// TIA Portal V16 export
// export: Created 2025-05-24T14:07:36.0860852Z, ExportSetting WithDefaults, DisplayName Totally Integrated Automation Portal, DisplayVersion V16, DisplayName TIA Portal Version Control Interface, DisplayVersion V16, DisplayName TIA Portal Openness, DisplayVersion V16, DisplayName STEP 7 Professional, DisplayVersion V16, DisplayName STEP 7 Safety, DisplayVersion V16, DisplayName WinCC Advanced, DisplayVersion V16
FUNCTION "6 - Storingsmelding" : Void   // FC8, LAD
TITLE = Warnings
VERSION : 0.1
// This program block is for audible & visual warnings.
// stored: AutoNumber true, IsIECCheckEnabled false, UDAEnableTagReadback false
   VAR_TEMP
      "Wals Sensor Controlled" : Bool;
      "Infeed Sensor Controlled" : Bool;
   END_VAR
   VAR CONSTANT
      "Sensor 2 (option)" : Bool := TRUE;
   END_VAR
   VAR_TEMP   // added for the SCL form of the ladder/FBD networks
      _w1 : Bool;
   END_VAR
BEGIN

REGION Network 1: +MC-21K6:5 - Bel Storing
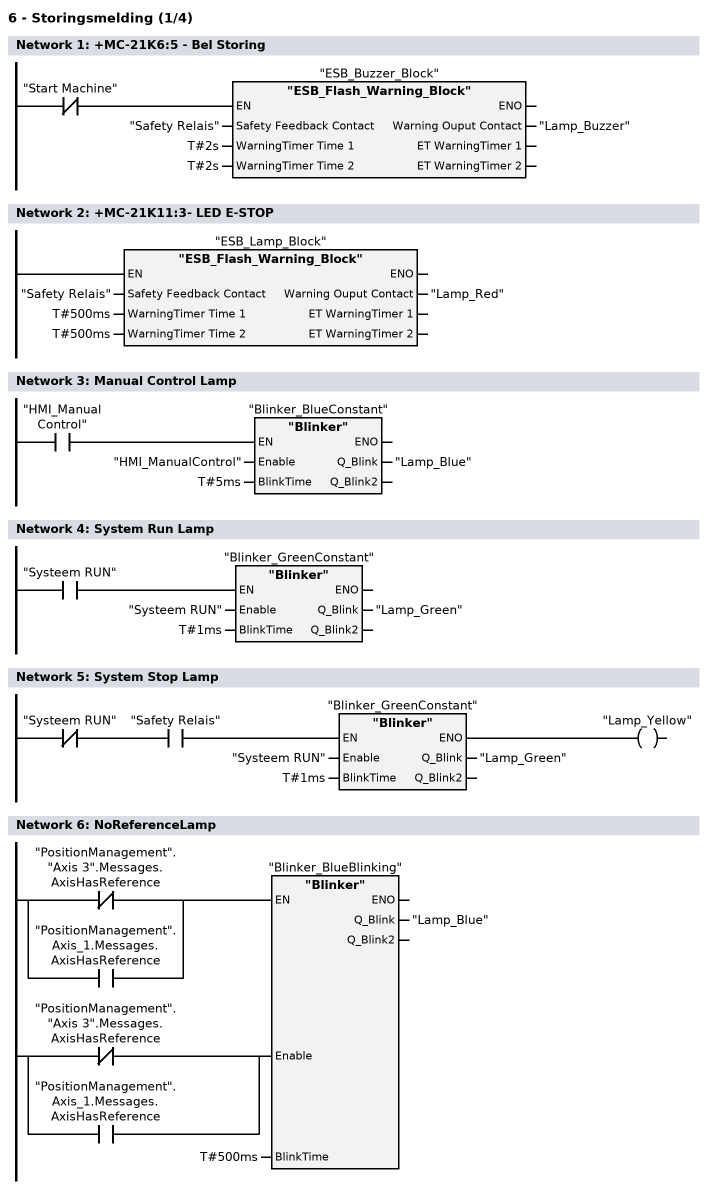
   RUNG wire#powerrail
      I_Contact( "Start Machine" )
      "ESB_Buzzer_Block"("Safety Feedback Contact" := "Safety Relais", "WarningTimer Time 1" := T#2s, "WarningTimer Time 2" := T#2s, "Warning Ouput Contact" => "Lamp_Buzzer", "ET WarningTimer 1" =>, "ET WarningTimer 2" =>)
   END_RUNG
   // the same network as SCL:
   IF NOT "Start Machine" THEN
       "ESB_Buzzer_Block"("Safety Feedback Contact" := "Safety Relais",   // "ESB_Flash_Warning_Block"
                          "WarningTimer Time 1" := T#2s,
                          "WarningTimer Time 2" := T#2s,
                          "Warning Ouput Contact" => "Lamp_Buzzer");
   END_IF;
END_REGION

REGION Network 2: +MC-21K11:3- LED E-STOP
   RUNG wire#powerrail
      "ESB_Lamp_Block"("Safety Feedback Contact" := "Safety Relais", "WarningTimer Time 1" := T#500ms, "WarningTimer Time 2" := T#500ms, "Warning Ouput Contact" => "Lamp_Red", "ET WarningTimer 1" =>, "ET WarningTimer 2" =>)
   END_RUNG
   // the same network as SCL:
   "ESB_Lamp_Block"("Safety Feedback Contact" := "Safety Relais",   // "ESB_Flash_Warning_Block"
                    "WarningTimer Time 1" := T#500ms,
                    "WarningTimer Time 2" := T#500ms,
                    "Warning Ouput Contact" => "Lamp_Red");
END_REGION

REGION Network 3: Manual Control Lamp
   RUNG wire#powerrail
      Contact( "HMI_ManualControl" )
      "Blinker_BlueConstant"(Enable := "HMI_ManualControl", BlinkTime := T#5ms, Q_Blink => "Lamp_Blue", Q_Blink2 =>)
   END_RUNG
   // the same network as SCL:
   IF "HMI_ManualControl" THEN
       "Blinker_BlueConstant"(Enable := "HMI_ManualControl", BlinkTime := T#5ms, Q_Blink => "Lamp_Blue");   // "Blinker"
   END_IF;
END_REGION

REGION Network 4: System Run Lamp
   RUNG wire#powerrail
      Contact( "Systeem RUN" )
      "Blinker_GreenConstant"(Enable := "Systeem RUN", BlinkTime := T#1ms, Q_Blink => "Lamp_Green", Q_Blink2 =>)
   END_RUNG
   // the same network as SCL:
   IF "Systeem RUN" THEN
       "Blinker_GreenConstant"(Enable := "Systeem RUN", BlinkTime := T#1ms, Q_Blink => "Lamp_Green");   // "Blinker"
   END_IF;
END_REGION

REGION Network 5: System Stop Lamp
   RUNG wire#powerrail
      I_Contact( "Systeem RUN" )
      Contact( "Safety Relais" )
      "Blinker_GreenConstant"(Enable := "Systeem RUN", BlinkTime := T#1ms, Q_Blink => "Lamp_Green", Q_Blink2 =>)
      Coil( "Lamp_Yellow" )
   END_RUNG
   // the same network as SCL:
   "Blinker_GreenConstant"(EN := NOT "Systeem RUN" AND "Safety Relais",   // "Blinker"
                           Enable := "Systeem RUN",
                           BlinkTime := T#1ms,
                           Q_Blink => "Lamp_Green",
                           ENO => #_w1);
   "Lamp_Yellow" := #_w1;
END_REGION

REGION Network 6: NoReferenceLamp
   RUNG wire#powerrail
      I_Contact( "PositionManagement"."Axis 3".Messages.AxisHasReference )
      wire#w1
      "Blinker_BlueBlinking"(Enable := wire#w2, BlinkTime := T#500ms, Q_Blink => "Lamp_Blue", Q_Blink2 =>)
   END_RUNG
   RUNG wire#powerrail
      Contact( "PositionManagement".Axis_1.Messages.AxisHasReference )
   END_RUNG wire#w1
   RUNG wire#powerrail
      I_Contact( "PositionManagement"."Axis 3".Messages.AxisHasReference )
   END_RUNG wire#w2
   RUNG wire#powerrail
      Contact( "PositionManagement".Axis_1.Messages.AxisHasReference )
   END_RUNG wire#w2
   // the same network as SCL:
   IF NOT "PositionManagement"."Axis 3".Messages.AxisHasReference OR "PositionManagement".Axis_1.Messages.AxisHasReference THEN
       "Blinker_BlueBlinking"(Enable := NOT "PositionManagement"."Axis 3".Messages.AxisHasReference OR "PositionManagement".Axis_1.Messages.AxisHasReference,   // "Blinker"
                              BlinkTime := T#500ms,
                              Q_Blink => "Lamp_Blue");
   END_IF;
END_REGION

REGION Network 7: Fill Trechter Delay Function
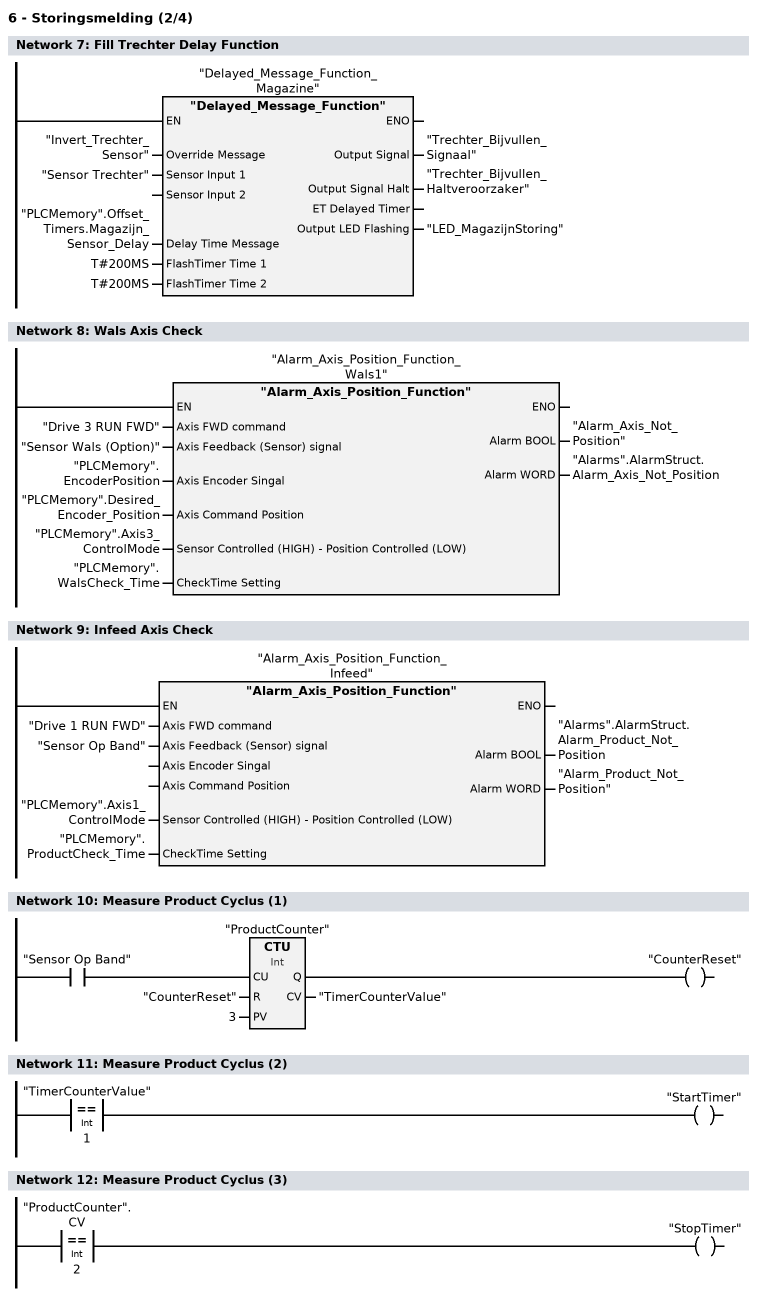
   RUNG wire#powerrail
      "Delayed_Message_Function_Magazine"("Override Message" := "Invert_Trechter_Sensor", "Sensor Input 1" := "Sensor Trechter", "Sensor Input 2" :=, "Delay Time Message" := "PLCMemory".Offset_Timers.Magazijn_Sensor_Delay, "FlashTimer Time 1" := T#200MS, "FlashTimer Time 2" := T#200MS, "Output Signal" => "Trechter_Bijvullen_Signaal", "Output Signal Halt" => "Trechter_Bijvullen_Haltveroorzaker", "ET Delayed Timer" =>, "Output LED Flashing" => "LED_MagazijnStoring")
   END_RUNG
   // the same network as SCL:
   "Delayed_Message_Function_Magazine"("Override Message" := "Invert_Trechter_Sensor",   // "Delayed_Message_Function"
                           "Sensor Input 1" := "Sensor Trechter",
                           "Delay Time Message" := "PLCMemory".Offset_Timers.Magazijn_Sensor_Delay,
                           "FlashTimer Time 1" := T#200MS,
                           "FlashTimer Time 2" := T#200MS,
                           "Output Signal" => "Trechter_Bijvullen_Signaal",
                           "Output Signal Halt" => "Trechter_Bijvullen_Haltveroorzaker",
                           "Output LED Flashing" => "LED_MagazijnStoring");
END_REGION

REGION Network 8: Wals Axis Check
   RUNG wire#powerrail
      "Alarm_Axis_Position_Function_Wals1"("Axis FWD command" := "Drive 3 RUN FWD", "Axis Feedback (Sensor) signal" := "Sensor Wals (Option)", "Axis Encoder Singal" := "PLCMemory".EncoderPosition, "Axis Command Position" := "PLCMemory".Desired_Encoder_Position, "Sensor Controlled (HIGH) - Position Controlled (LOW)" := "PLCMemory".Axis3_ControlMode, "CheckTime Setting" := "PLCMemory".WalsCheck_Time, "Alarm BOOL" => "Alarm_Axis_Not_Position", "Alarm WORD" => "Alarms".AlarmStruct.Alarm_Axis_Not_Position)
   END_RUNG
   // the same network as SCL:
   "Alarm_Axis_Position_Function_Wals1"("Axis FWD command" := "Drive 3 RUN FWD",   // "Alarm_Axis_Position_Function"
                           "Axis Feedback (Sensor) signal" := "Sensor Wals (Option)",
                           "Axis Encoder Singal" := "PLCMemory".EncoderPosition,
                           "Axis Command Position" := "PLCMemory".Desired_Encoder_Position,
                           "Sensor Controlled (HIGH) - Position Controlled (LOW)" := "PLCMemory".Axis3_ControlMode,
                           "CheckTime Setting" := "PLCMemory".WalsCheck_Time,
                           "Alarm BOOL" => "Alarm_Axis_Not_Position",
                           "Alarm WORD" => "Alarms".AlarmStruct.Alarm_Axis_Not_Position);
END_REGION

REGION Network 9: Infeed Axis Check
   RUNG wire#powerrail
      "Alarm_Axis_Position_Function_Infeed"("Axis FWD command" := "Drive 1 RUN FWD", "Axis Feedback (Sensor) signal" := "Sensor Op Band", "Axis Encoder Singal" :=, "Axis Command Position" :=, "Sensor Controlled (HIGH) - Position Controlled (LOW)" := "PLCMemory".Axis1_ControlMode, "CheckTime Setting" := "PLCMemory".ProductCheck_Time, "Alarm BOOL" => "Alarms".AlarmStruct.Alarm_Product_Not_Position, "Alarm WORD" => "Alarm_Product_Not_Position")
   END_RUNG
   // the same network as SCL:
   "Alarm_Axis_Position_Function_Infeed"("Axis FWD command" := "Drive 1 RUN FWD",   // "Alarm_Axis_Position_Function"
                           "Axis Feedback (Sensor) signal" := "Sensor Op Band",
                           "Sensor Controlled (HIGH) - Position Controlled (LOW)" := "PLCMemory".Axis1_ControlMode,
                           "CheckTime Setting" := "PLCMemory".ProductCheck_Time,
                           "Alarm BOOL" => "Alarms".AlarmStruct.Alarm_Product_Not_Position,
                           "Alarm WORD" => "Alarm_Product_Not_Position");
END_REGION

REGION Network 10: Measure Product Cyclus (1)
   RUNG wire#powerrail
      Contact( "Sensor Op Band" )
      { S7_Templates := "value_type := Int" } "ProductCounter".CTU(r := "CounterReset", pv := 3, cv => "TimerCounterValue")
      Coil( "CounterReset" )
   END_RUNG
   // the same network as SCL:
   "ProductCounter".CTU(CU := "Sensor Op Band", R := "CounterReset", PV := 3, CV => "TimerCounterValue");
   "CounterReset" := "ProductCounter".Q;
END_REGION

REGION Network 11: Measure Product Cyclus (2)
   RUNG wire#powerrail
      { S7_Templates := "SrcType := Int" } EQ_Contact(in1 := "TimerCounterValue", in2 := 1)
      Coil( "StartTimer" )
   END_RUNG
   // the same network as SCL:
   "StartTimer" := "TimerCounterValue" = 1;
END_REGION

REGION Network 12: Measure Product Cyclus (3)
   RUNG wire#powerrail
      { S7_Templates := "SrcType := Int" } EQ_Contact(in1 := "ProductCounter".CV, in2 := 2)
      Coil( "StopTimer" )
   END_RUNG
   // the same network as SCL:
   "StopTimer" := "ProductCounter".CV = 2;
END_REGION

REGION Network 13: Measure Product Cyclus (4)
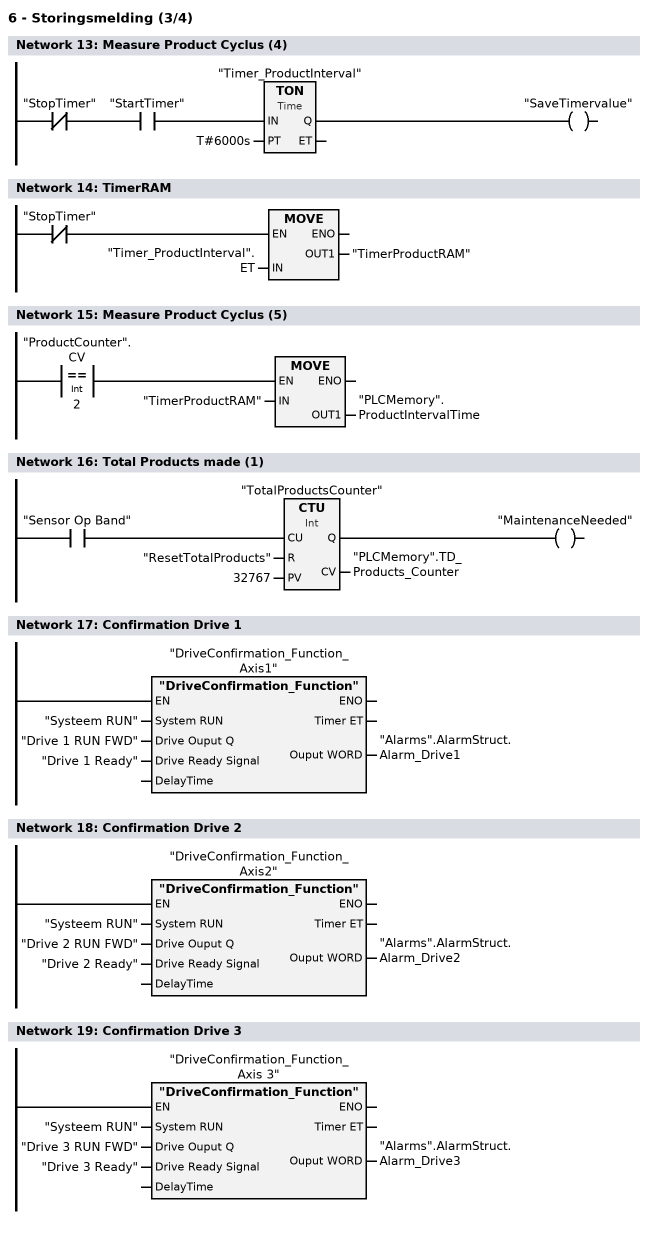
   RUNG wire#powerrail
      I_Contact( "StopTimer" )
      Contact( "StartTimer" )
      { S7_Templates := "time_type := Time" } "Timer_ProductInterval".TON(pt := T#6000s, et =>)
      Coil( "SaveTimervalue" )
   END_RUNG
   // the same network as SCL:
   "Timer_ProductInterval".TON(IN := NOT "StopTimer" AND "StartTimer", PT := T#6000s);
   "SaveTimervalue" := "Timer_ProductInterval".Q;
END_REGION

REGION Network 14: TimerRAM
   RUNG wire#powerrail
      I_Contact( "StopTimer" )
      { S7_GenerateENO := "TRUE" } Move(in := "Timer_ProductInterval".ET, out1 => "TimerProductRAM")
   END_RUNG
   // the same network as SCL:
   IF NOT "StopTimer" THEN "TimerProductRAM" := "Timer_ProductInterval".ET; END_IF;
END_REGION

REGION Network 15: Measure Product Cyclus (5)
   RUNG wire#powerrail
      { S7_Templates := "SrcType := Int" } EQ_Contact(in1 := "ProductCounter".CV, in2 := 2)
      { S7_GenerateENO := "TRUE" } Move(in := "TimerProductRAM", out1 => "PLCMemory".ProductIntervalTime)
   END_RUNG
   // the same network as SCL:
   IF "ProductCounter".CV = 2 THEN "PLCMemory".ProductIntervalTime := "TimerProductRAM"; END_IF;
END_REGION

REGION Network 16: Total Products made (1)
   RUNG wire#powerrail
      Contact( "Sensor Op Band" )
      { S7_Templates := "value_type := Int" } "TotalProductsCounter".CTU(r := "ResetTotalProducts", pv := 32767, cv => "PLCMemory".TD_Products_Counter)
      Coil( "MaintenanceNeeded" )
   END_RUNG
   // the same network as SCL:
   "TotalProductsCounter".CTU(CU := "Sensor Op Band",
                           R := "ResetTotalProducts",
                           PV := 32767,
                           CV => "PLCMemory".TD_Products_Counter);
   "MaintenanceNeeded" := "TotalProductsCounter".Q;
END_REGION

REGION Network 17: Confirmation Drive 1
   RUNG wire#powerrail
      "DriveConfirmation_Function_Axis1"("System RUN" := "Systeem RUN", "Drive Ouput Q" := "Drive 1 RUN FWD", "Drive Ready Signal" := "Drive 1 Ready", DelayTime :=, "Timer ET" =>, "Ouput WORD" => "Alarms".AlarmStruct.Alarm_Drive1)
   END_RUNG
   // the same network as SCL:
   "DriveConfirmation_Function_Axis1"("System RUN" := "Systeem RUN",   // "DriveConfirmation_Function"
                           "Drive Ouput Q" := "Drive 1 RUN FWD",
                           "Drive Ready Signal" := "Drive 1 Ready",
                           "Ouput WORD" => "Alarms".AlarmStruct.Alarm_Drive1);
END_REGION

REGION Network 18: Confirmation Drive 2
   RUNG wire#powerrail
      "DriveConfirmation_Function_Axis2"("System RUN" := "Systeem RUN", "Drive Ouput Q" := "Drive 2 RUN FWD", "Drive Ready Signal" := "Drive 2 Ready", DelayTime :=, "Timer ET" =>, "Ouput WORD" => "Alarms".AlarmStruct.Alarm_Drive2)
   END_RUNG
   // the same network as SCL:
   "DriveConfirmation_Function_Axis2"("System RUN" := "Systeem RUN",   // "DriveConfirmation_Function"
                           "Drive Ouput Q" := "Drive 2 RUN FWD",
                           "Drive Ready Signal" := "Drive 2 Ready",
                           "Ouput WORD" => "Alarms".AlarmStruct.Alarm_Drive2);
END_REGION

REGION Network 19: Confirmation Drive 3
   RUNG wire#powerrail
      "DriveConfirmation_Function_Axis 3"("System RUN" := "Systeem RUN", "Drive Ouput Q" := "Drive 3 RUN FWD", "Drive Ready Signal" := "Drive 3 Ready", DelayTime :=, "Timer ET" =>, "Ouput WORD" => "Alarms".AlarmStruct.Alarm_Drive3)
   END_RUNG
   // the same network as SCL:
   "DriveConfirmation_Function_Axis 3"("System RUN" := "Systeem RUN",   // "DriveConfirmation_Function"
                           "Drive Ouput Q" := "Drive 3 RUN FWD",
                           "Drive Ready Signal" := "Drive 3 Ready",
                           "Ouput WORD" => "Alarms".AlarmStruct.Alarm_Drive3);
END_REGION

REGION Network 20: Confimation Drive 4
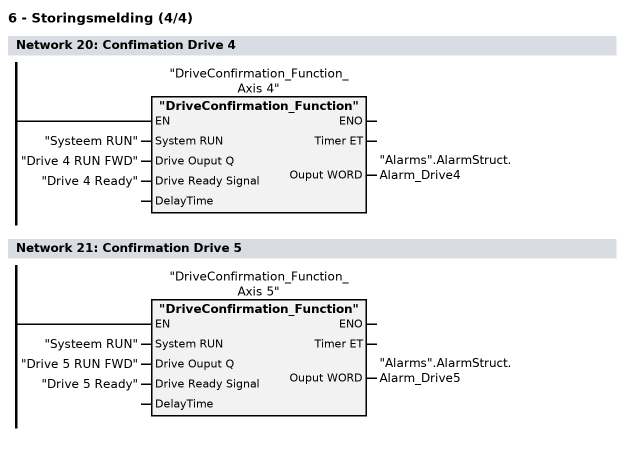
   RUNG wire#powerrail
      "DriveConfirmation_Function_Axis 4"("System RUN" := "Systeem RUN", "Drive Ouput Q" := "Drive 4 RUN FWD", "Drive Ready Signal" := "Drive 4 Ready", DelayTime :=, "Timer ET" =>, "Ouput WORD" => "Alarms".AlarmStruct.Alarm_Drive4)
   END_RUNG
   // the same network as SCL:
   "DriveConfirmation_Function_Axis 4"("System RUN" := "Systeem RUN",   // "DriveConfirmation_Function"
                           "Drive Ouput Q" := "Drive 4 RUN FWD",
                           "Drive Ready Signal" := "Drive 4 Ready",
                           "Ouput WORD" => "Alarms".AlarmStruct.Alarm_Drive4);
END_REGION

REGION Network 21: Confirmation Drive 5
   RUNG wire#powerrail
      "DriveConfirmation_Function_Axis 5"("System RUN" := "Systeem RUN", "Drive Ouput Q" := "Drive 5 RUN FWD", "Drive Ready Signal" := "Drive 5 Ready", DelayTime :=, "Timer ET" =>, "Ouput WORD" => "Alarms".AlarmStruct.Alarm_Drive5)
   END_RUNG
   // the same network as SCL:
   "DriveConfirmation_Function_Axis 5"("System RUN" := "Systeem RUN",   // "DriveConfirmation_Function"
                           "Drive Ouput Q" := "Drive 5 RUN FWD",
                           "Drive Ready Signal" := "Drive 5 Ready",
                           "Ouput WORD" => "Alarms".AlarmStruct.Alarm_Drive5);
END_REGION
END_FUNCTION
